(*
  Specific printhead implementing the grid logic.
*)
FUNCTION_BLOCK FB_PH_Grid EXTENDS FB_PH IMPLEMENTS I_Correction_Grid
VAR
  // fifo queue
  fbFifo            : FB_GridPointFIFO;    // points fifo
  
  // queue status
  _bQueueBusy       : BOOL;               // point queue is not empty
  _bQueueError      : BOOL;               // point queue has an error

  // grid settings
  _bGridSet         : BOOL;               // grid is configured
  _nRows            : DINT;               // number of roi rows
  _nRowLowerBound, _nRowUpperBound : DINT;  //limites for roi rows of this ph
  _sDefGridSettings : ST_DefGridSettings;  // grid settings
  
  // checks
  _fbGetTaskIdx     : GETCURTASKINDEX;
  _taskIdx          : UDINT;
  _sTaskInfo        : PlcTaskSystemInfo;
  _lastCycle        : UDINT;
    
  // debug
  bEnSimPoints      : BOOL;               // enable grid point simulation
  bEnDebug          : BOOL;               // enable grid point history & point dump in logger
  nPointHead        : INT := 0;           // last list entry
  sPointHistory     : ARRAY[0..100] OF ST_GridPoint; // grid point history array
END_VAR

// sync points fifo to CB (PHs)
syncPoints();

// debug
IF bEnSimPoints THEN simPoints(); END_IF

PROPERTY bPointQueueBusy : BOOL
GET
bPointQueueBusy := SEL(fbFifo.nCount>0, FALSE, TRUE);   // busy as long queue is not empty
END_GET
END_PROPERTY

PROPERTY bPointQueueError : BOOL
GET
// check for errors
IF fbFifo.bError THEN
  _bQueueError := TRUE;
ELSE
  bPointQueueError := FALSE;
END_IF
END_GET
END_PROPERTY

(*
  Convert a point from DefGrid point to a GridPoint for hw write.
*)
METHOD PRIVATE convertPoint : ST_GridPoint
VAR_INPUT
  sPoint : POINTER TO ST_DeformationPoint;
  nPhPosY : DINT;
END_VAR
VAR
  nRoiOffset : DINT;
END_VAR
IF _sDefGridSettings.nGridPitchY = 0 THEN F_Report_Error(ErrType:=EN_REPORT_ERROR_TYPE.Report_Error_0Pointer); RETURN; END_IF

convertPoint.dx := DINT_TO_UINT(sPoint^.dx);
convertPoint.dy := DINT_TO_UINT(sPoint^.dy);

// variant1 with absolute Node address (based on number of grid-rows
(*convertPoint.node := 
  UDINT_TO_UINT(
      DINT_TO_UDINT(sPoint^.col)*sDefGridSettings.nGridSizeY 
    + DINT_TO_UDINT(sPoint^.row)
);*)

// variant2 - calculate FPGA ROI_address (roi_buffer address of grid point)
{warning 'TODO: update constants for calculation if FPGA is ok and make CONSTANTS'}
nRoiOffset := nPhPosY / TO_DINT(_sDefGridSettings.nGridPitchY);
convertPoint.node := TO_UINT((sPoint^.col MOD GVL_Deformation.nC_GridRoiCols) * GVL_Deformation.nC_GridRoiRows + sPoint^.row - nRoiOffset);
END_METHOD

(*
  Keep a history of last synced points.
*)
METHOD PRIVATE history
VAR_INPUT
  pPoint  : POINTER TO ST_GridPoint;
END_VAR
IF pPoint^.node = 0 THEN nPointHead := 0; END_IF  // internal reset on point address 0

sPointHistory[nPointHead] := pPoint^;
nPointHead := (nPointHead + 1) MOD 100;
END_METHOD

METHOD init : BOOL
VAR_INPUT
  pAdsIf        : POINTER TO ST_ADS_PH;                (*Pointer to its ads interface structure*)
  sPhDef        : ST_PH_DEF;                           (*ph definition structure*)
  tTempMonitor  : TIME;                                (*ph temperature monitoring timeout (warning after elapsed time)*)
END_VAR
VAR
  bErr          : BOOL;
END_VAR
SUPER^.init(
    pAdsIf:=pAdsIf,
    sPhDef:=sPhDef,
    tTempMonitor:=tTempMonitor
);

nCorrection := 0;

_fbGetTaskIdx();
_taskIdx := _fbGetTaskIdx.index;
END_METHOD

(*
  Configure grid settings for ph.
*)
METHOD setGrid
VAR_INPUT
  sGrid : ST_DefGridSettings;
END_VAR
// grid settings checks
IF sGrid.nGridPitchX = 0 OR sGrid.nGridPitchY = 0 OR sGrid.nGridPoints = 0 THEN
  LogError('Invalid grid settings');
  RETURN;
END_IF

// store grid settings
_sDefGridSettings :=sGrid;

// caluclate roi row bounds
// lower row bound
_nRowLowerBound:=nPositionY / UDINT_TO_DINT(_sDefGridSettings.nGridPitchY);   // floor
_nRowLowerBound := LIMIT(0, _nRowLowerBound, UDINT_TO_DINT(_sDefGridSettings.nGridSizeY));  // limit to grid scope

// upper row bound
_nRowUpperBound:=(nPositionY + nHeadWidth) / UDINT_TO_DINT(_sDefGridSettings.nGridPitchY) + 1;
_nRowUpperBound := LIMIT(0, _nRowUpperBound, UDINT_TO_DINT(_sDefGridSettings.nGridSizeY));  // limit to grid scope

{warning 'TODO: update if RIO requirements are set by FPGA'}
// we just force to have 4 ROI rows and always charge effectively 4 row per head event if 3 would be sufficent
_nRowUpperBound := _nRowLowerBound + GVL_Deformation.nC_GridRoiRows - 1; 
// number of rows
_nRows := _nRowUpperBound - _nRowLowerBound + 1;

_bGridSet := TRUE;
END_METHOD

METHOD PRIVATE simPoints
VAR_INST
  tWrPoint      : TON := (PT:=T#1S);
  RandomNumber  : DRAND;
  sGridCfg    : ST_DefGridSettings := (nGridPitchX:=1024, nGridPitchY:=1024, nGridSizeX:=100, nGridSizeY:=100, nGridPoints:=10_000, nGridImageOffsetY:=0);   // some simulation defaults
  sNewPoint   : ST_DeformationPoint;
END_VAR
VAR
  random_val  : LREAL;
END_VAR
IF NOT _bGridSet THEN setGrid(sGrid:=sGridCfg); END_IF

// create and write a
tWrPoint(IN:=NOT tWrPoint.Q);
IF tWrPoint.Q THEN
  RandomNumber(Seed:=12, Num=>random_val);
  sNewPoint.dx := DINT_TO_UINT(FC_LREAL_TO_DINT((random_val * 100) - 50));
  RandomNumber(Seed:=12, Num=>random_val);
  sNewPoint.dy := DINT_TO_UINT(FC_LREAL_TO_DINT((random_val * 60) - 30));
  sNewPoint.col := sNewPoint.index / _nRows;
  sNewPoint.row := sNewPoint.index MOD _nRows + _nRowLowerBound;
  sNewPoint.index := (sNewPoint.index + 1) MOD 20;  // just 20 points
  writeCorrectionPoint(sPoint:=sNewPoint);
END_IF
END_METHOD

(*
  Sync deformation point to hardware.
*)
METHOD PRIVATE syncPoints
VAR
  sPoint  : ST_GridPoint;
  bOK     : BOOL;
  nPdiVal : ULINT;
END_VAR

IF fbFifo.nCount > 0 THEN
  bOK := fbFifo.Pop(sGridPoint=>sPoint);
  IF bOK THEN
    // build grid point pdi data
    nPdiVal     := UINT_TO_ULINT(sPoint.dx);
    nPdiVal     := nPdiVal OR SHL(UINT_TO_ULINT(sPoint.dy), 16);
    nPdiVal     := nPdiVal OR SHL(UINT_TO_ULINT(sPoint.node), 32);  
  
    sendCorrection(nCmdBit:=nC_CORRECTION_CMDBIT_GRIDPOINT, nData:=nPdiVal);

    //history
    IF bEnable AND bEnDebug THEN history(ADR(sPoint)); END_IF
  ELSE
    LogError('syncPoints: could not get a new GridPoint');
	END_IF
END_IF

// check for double calls within one task cycle
_sTaskInfo := TwinCAT_SystemInfoVarList._TaskInfo[_taskIdx];
IF _sTaskInfo.CycleCount = _lastCycle THEN
  LogError('syncPoints: was called twice in same task cycle');
END_IF
_lastCycle := _sTaskInfo.CycleCount;
END_METHOD

METHOD PRIVATE syncPoints_old
VAR
  sPoint  : ST_GridPoint;
  bOK     : BOOL;
  nPdiVal : ULINT;
END_VAR
nCorrection := nCorrection AND 16#0000FFFFFFFFFFFF;  // reset correction command only

IF fbFifo.nCount > 0 THEN
  bOK := fbFifo.Pop(sGridPoint=>sPoint);
  IF bOK THEN
    // build grid point pdi data
    nPdiVal     := UINT_TO_ULINT(sPoint.dx);
    nPdiVal     := nPdiVal OR SHL(UINT_TO_ULINT(sPoint.dy), 16);
    nPdiVal     := nPdiVal OR SHL(UINT_TO_ULINT(sPoint.node), 32);  
  
    // old sending (direct nCorrection access
    nCorrection := nCorrection AND 16#0000FFFFFFFFFFFF;  // reset correction command only
    nCorrection := SHL(1, 48) OR nPdiVal;      //set cmd [16bit] cmd / [48bit] of grid point in PDI var

    //history
    IF bEnable AND bEnDebug THEN history(ADR(sPoint)); END_IF
  ELSE
    LogError('syncPoints: could not get a new GridPoint');
	END_IF
END_IF
END_METHOD

(*
  Write a new Deformation Point to the hardware. 
  New added points will be synchroniced with the hardware with a FIFO queue.
  :return: TRUE on success
*)
METHOD writeCorrectionPoint : BOOL
VAR_INPUT
	(* add a new deformation point*)
	sPoint	: ST_DeformationPoint;
END_VAR
VAR
  sGridPoint : ST_GridPoint;
END_VAR
IF NOT _bGridSet THEN RETURN; END_IF

// filter points only for this head
IF sPoint.row >= _nRowLowerBound AND sPoint.row <= _nRowUpperBound THEN
  
  // convert deformation point to GridPoint for hw
  sGridPoint := convertPoint(sPoint:=ADR(sPoint), nPositionY);
  
  // add point
  writeCorrectionPoint := fbFifo.Push(sNewPoint:=sGridPoint);   // add new point

  IF bEnable AND bEnDebug THEN
    LogLvl(Lvl:=E_LogSeverity.Debug, Msg:=
      F_Concat4(
        'Write GridPoint '
        ,F_Concat4('c:', TO_STRING(sPoint.col), ' r:', TO_STRING(sPoint.row))
        ,F_Concat2(' -> node:', TO_STRING(sGridPoint.node))
        ,F_Concat4(' dx:', TO_STRING(sPoint.dx), ' dy:', TO_STRING(sPoint.dy))
      )
    );
  END_IF

END_IF
END_METHOD

END_FUNCTION_BLOCK

(* stored: Version 1.1.0.1, ProductVersion 3.1.4024.11
   POU FB_PH_Grid: Id {7d84493e-c0db-481a-b913-ca603f9217d7}, SpecialFunc None
   Property bPointQueueBusy: Id {743cb526-13a9-4a34-8340-5ce273e1a04d}
   Get Get: Id {042e433e-239b-4c3d-b0fd-109113d4f688}
   Property bPointQueueError: Id {15f61a7e-74db-4c93-8e7b-82ebe5f7fac2}
   Get Get: Id {1b0e0081-4894-40c9-9088-5c494fb1f80a}
   Method convertPoint: Id {ce218d93-eaab-4eb2-903f-9bc8545e9f37}
   Method history: Id {51c013f7-5b60-4957-af19-f90b1fe2cb67}
   Method init: Id {aac88526-a64d-4341-b09a-21e8f02199be}
   Method setGrid: Id {b19c3f25-5f02-485e-a505-24a5847f95da}
   Method simPoints: Id {6c01aed3-a0eb-4fe3-8ba0-4a6c5b8f59ed}
   Method syncPoints: Id {d34e75ef-e0c7-4871-9b57-12d9c3403c8e}
   Method syncPoints_old: Id {5eb58362-cb73-42e8-a336-d248e00b91f9}
   Method writeCorrectionPoint: Id {a049beb6-fde3-4da4-ba01-912d4c21c5c6} *)
